Staubli VAL3: _displayList.pgx

program _displayList(string x_sDirectory (dimensions=1), string x_sTitle (dimensions=1), num x_nX (dimensions=1), num x_nY (dimensions=1), num x_nWidth (dimensions=1), num x_nHeight (dimensions=1))
  local num l_i
begin
  // This program explores a directory, generates and display
  // a list with the files included in that directory
  //
  // Input Param
  // x_sDirectory : Directory to explore
  //
  // Output Param
  //  x_nError    : Error code
  //
  // Created 23-02-05                                   C.CURRIVAND
  //----------------------------------------------------------------
  // Resize variable
  resize(sItemList,1,1)
  //
  call up:listSetSize(x_nX,x_nY,x_nWidth,x_nHeight)
  call up:listCreate(x_sTitle)
  if libList(x_sDirectory,sItemList)==true
    call up:listAdd(sItemList)
    call up:listUpdate(0)
  endIf
end
